{attribute 'linkalways'} 
{attribute 'no_explicit_call' := 'This FB is a CLASS and must be accessed using methods or properties'}
{attribute 'enable_dynamic_creation'}
FUNCTION_BLOCK Node_RGBA_WHITE EXTENDS VisionNode
VAR
    out : _TcVnVector4_LREAL;
END_VAR

METHOD PUBLIC  Clone : I_Node
VAR
	pNode : POINTER TO Node_RGBA_WHITE;
END_VAR
pNode := __NEW(Node_RGBA_WHITE);
Clone := pNode^;
END_METHOD

METHOD FB_init : BOOL
VAR_INPUT
	bInitRetains : BOOL; // if TRUE, the retain variables are initialized (warm start / cold start)
	bInCopyCode : BOOL;  // if TRUE, the instance afterwards gets moved into the copy code (online change)
END_VAR
AddOutput('out', out);
END_METHOD

METHOD PROTECTED OnExecute
out.Value := GVL_COLOURS.RGBA_WHITE;
END_METHOD

METHOD PUBLIC PreExecutionCheck
VAR_INPUT
	Check : I_PreExecutionChecks;
END_VAR
END_METHOD

END_FUNCTION_BLOCK

(* stored: Version 1.1.0.1, ProductVersion 3.1.4024.13
   POU Node_RGBA_WHITE: Id {793a0e40-2760-0401-0bc9-57ead7efea25}, SpecialFunc None
   Folder Constructor: Id {a396dd87-ac2c-0ce1-29c0-9b50ff3ed5b6}
   Method Clone: Id {14848323-feac-0131-34d1-05d5d5115ad9}
   Method FB_init: Id {13b64325-dc67-055c-08e7-baec7a345c5f}
   Method OnExecute: Id {4c226fe2-66f1-0dd3-2f3d-6fbe747d590b}
   Method PreExecutionCheck: Id {e5d5cfc1-e2b3-0d69-294f-f96206271425} *)
